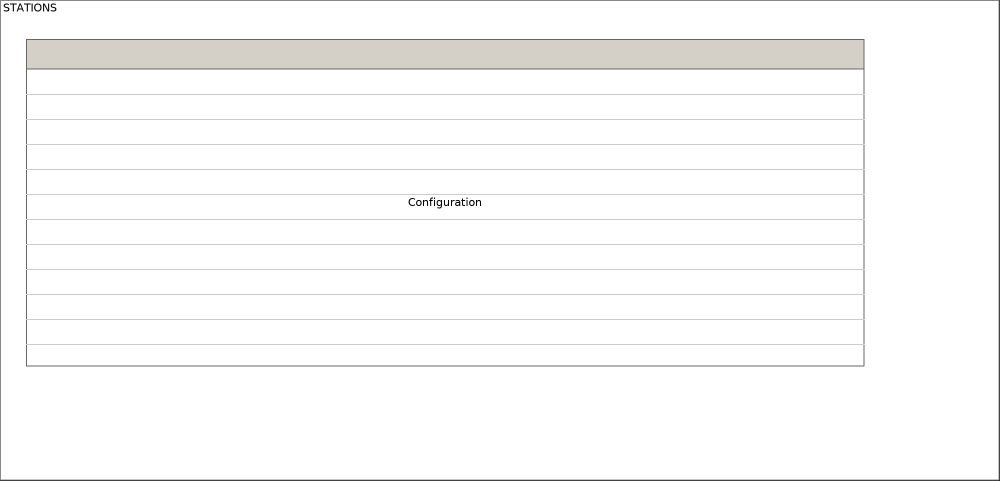
VISUALIZATION VI_XTSStationsVisu  // 1000x481
VAR_IN_OUT
	xts : XTS_System;
END_VAR
VAR
	stTableStruct : ARRAY [1..25] OF stTableStructx10;
END_VAR
    Rectangle (0,0 1000x481), "STATIONS"
    Table (26,39 838x327), "Configuration", data array: stTableStruct
        p3854506369: xts.stCfg.stStationsCfg[INDEX].sName
        p1892666644: xts.stCfg.stStationsCfg[INDEX].bEnableManualAck
        p338671338: xts.stCfg.stStationsCfg[INDEX].bManualAck
        p2170511999: xts.aStations[INDEX].fbMoversFIFO.nMovers
        p3723444502: xts.aStations[INDEX].udiSequenceState
        p1218418051: xts.aStations[INDEX].udiErrorID
        p746581629: xts.aStations[INDEX].sMoversWaiting
        p3104783080: xts.aStations[INDEX].sMoversIn
        p7306298: xts.stCfg.stStationsCfg[INDEX].lrEndPosition
        p511219082: Manual Ack
        p4092479075: Movers Waiting
        p505689113: Error ID
        p4088588272: Movers In
        p2243050616: Extra Cfg.
        p516019884: End Position
        p2685023577: stTableStruct.b1
        p3312258591: stTableStruct.b2
        p1791247317: stTableStruct.b3
        p262371475: stTableStruct.b4
        p4008173056: stTableStruct.b5
        p2340480326: stTableStruct.b6
        p606709900: stTableStruct.b7
        p1095668682: stTableStruct.b8
        p1037165547: stTableStruct.b9
        p1488378029: stTableStruct.b10
        Columns.Column.[3].Template: xts.aStations[INDEX].bWaitingMovers
        Columns.Column.[9].Template: OnMouseClick: write the text variable via Default
        Columns.Column.[6].Template: OnMouseClick: write the text variable via Default, min 1, max 3
        Columns.Column.[4].Template: OnMouseClick: write the text variable via Default
        Columns.Column.[5].Template: OnMouseClick: write the text variable via Default
        Columns.Column.[2].Template: tap xts.stCfg.stStationsCfg[INDEX].bManualAck
        Columns.Column.[0].Template: OnMouseClick: write the text variable via Default
        Columns.Column.[1].Template: toggle xts.stCfg.stStationsCfg[INDEX].bEnableManualAck
        Columns.Column.[7].Template: OnMouseClick: write the text variable via Default
END_VISUALIZATION

(* stored: Version 1.1.0.1, ProductVersion 3.1.4024.11
   Visu VI_XTSStationsVisu: Id {d4f05308-034f-4067-a730-7bcc926184bb} *)
